// TIA Portal project "PID_controller" (V14)

(* hardware
DEVICE "S71500/ET200MP station_1"  S7-1500 station
   slot 0: "Rail_0"  Rack  6ES7 590-1***0-0AA0
   slot 1: "SERVER_PID"  CPU 1512C-1 PN  6ES7 512-1CK00-0AB0  V2.1
      slot 3: "CPU display_1"  6ES7591-1AA00-0AA0
DEVICE "PID_HMI"  KTP700 Basic PN
   slot 0: "KTP700 Basic PN"  KTP700 Basic PN  6AV2 123-2GB03-0AX0  14.0.1.0
   slot 1: "HMI_RT_1"  KTP700 Basic PN  6AV2 123-2GB03-0AX0  14.0.1.0
   slot 5: "PID_HMI.IE_CP_1"  PROFINET Interface  14.0.1.0
      slot 1: "PROFINET Interface_1"  PROFINET Interface
         slot 1: "Port_1"  Port
*)

// ===== PLC "SERVER_PID"  CPU 1512C-1 PN =====

VAR_GLOBAL   // PLC tag table "Default tag table"
   "Temperature_input" AT %IW0 : Int;
   "Pump_out" AT %QW0 : Int;
END_VAR

DATA_BLOCK "Temperature"   // DB2
{ S7_Optimized_Access := 'TRUE' }
VERSION : 0.1
   VAR
      Temperature_input : Real;
      Temperature_out : Real;
   END_VAR
BEGIN
END_DATA_BLOCK

DATA_BLOCK "PID_DB"   // DB3
{ S7_Optimized_Access := 'TRUE' }
VERSION : 0.1
   VAR
      PID_Setpoint : Real;
      PID_Output : Real;
      PIT_Output_PER : Int;
      PId_Output_PWM : Bool;
      PID_State : Int;
      PID_Error : Bool;
      PID_ModeActivate : Bool;
      PID_manualEnable : Bool;
      PID_ErrorBits : Word;
   END_VAR
BEGIN
END_DATA_BLOCK

DATA_BLOCK "input_PLC_DB"   // DB4
{ S7_Optimized_Access := 'TRUE' }
VERSION : 0.1
// stored: InstanceOfName input_PLC
"input_PLC"
BEGIN
END_DATA_BLOCK

DATA_BLOCK "Pump_freuenceHz"   // DB5
{ S7_Optimized_Access := 'TRUE' }
VERSION : 0.1
   VAR
      Pump_scale : Real;
   END_VAR
BEGIN
END_DATA_BLOCK

FUNCTION_BLOCK "input_PLC"   // FB1, LAD
{ S7_Optimized_Access := 'TRUE' }
VERSION : 0.1
   VAR_INPUT
      input_plc : Real;
   END_VAR
   VAR_OUTPUT
      In_out_DB : Real;
   END_VAR
BEGIN

REGION Network 1
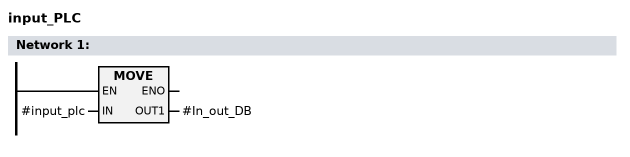
   RUNG wire#powerrail
      Move(in := #input_plc, out1 => #In_out_DB)
   END_RUNG
   // the same network as SCL:
   #In_out_DB := #input_plc;
END_REGION
END_FUNCTION_BLOCK

FUNCTION "analog_input" : Void   // FC1, LAD
{ S7_Optimized_Access := 'TRUE' }
VERSION : 0.1
   VAR_INPUT
      Inpit_min : Int;
      input_max : Int;
      Process_value : Real;
   END_VAR
   VAR_OUTPUT
      Scale_value_out : Real;
   END_VAR
   VAR_TEMP
      temp_value : Real;
   END_VAR
BEGIN

REGION Network 1
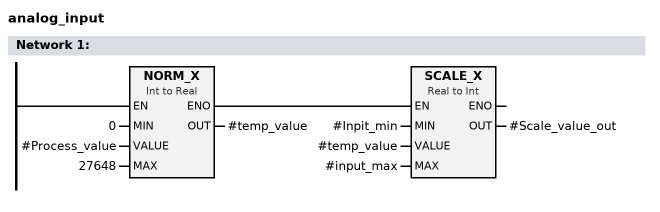
   RUNG wire#powerrail
      { S7_Templates := "[SrcType := Int, DestType := Real]" } Normalize(min := 0, value := #Process_value, max := 27648, out => #temp_value)
      { S7_Templates := "[SrcType := Real, DestType := Int]" } Scale(min := #Inpit_min, value := #temp_value, max := #input_max, out => #Scale_value_out)
   END_RUNG
   // the same network as SCL:
   #temp_value := NORM_X(MIN := 0, VALUE := #Process_value, MAX := 27648);
   #Scale_value_out := SCALE_X(MIN := #Inpit_min, VALUE := #temp_value, MAX := #input_max);
END_REGION
END_FUNCTION

ORGANIZATION_BLOCK "Main"   // OB1, LAD, ProgramCycle
TITLE = "Main Program Sweep (Cycle)"
{ S7_Optimized_Access := 'TRUE' }
VERSION : 0.1
   VAR_INPUT
      Initial_Call : Bool;   // Initial call of this OB
      Remanence : Bool;   // =True, if remanent data are available
   END_VAR
BEGIN

REGION Network 1
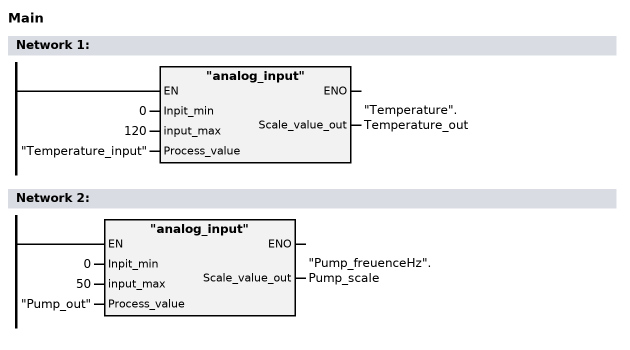
   RUNG wire#powerrail
      "analog_input"(Inpit_min := 0, input_max := 120, Process_value := "Temperature_input", Scale_value_out => "Temperature".Temperature_out)
   END_RUNG
   // the same network as SCL:
   "analog_input"(Inpit_min := 0,
                  input_max := 120,
                  Process_value := "Temperature_input",
                  Scale_value_out => "Temperature".Temperature_out);
END_REGION

REGION Network 2
   RUNG wire#powerrail
      "analog_input"(Inpit_min := 0, input_max := 50, Process_value := "Pump_out", Scale_value_out => "Pump_freuenceHz".Pump_scale)
   END_RUNG
   // the same network as SCL:
   "analog_input"(Inpit_min := 0,
                  input_max := 50,
                  Process_value := "Pump_out",
                  Scale_value_out => "Pump_freuenceHz".Pump_scale);
END_REGION
END_ORGANIZATION_BLOCK

ORGANIZATION_BLOCK "Cyclic interrupt"   // OB30, LAD, CyclicInterrupt
{ S7_Optimized_Access := 'TRUE' }
VERSION : 0.1
   VAR_INPUT
      Initial_Call : Bool;   // Initial call of this OB
      Event_Count : Int;   // Events discarded
   END_VAR
BEGIN

REGION Network 1
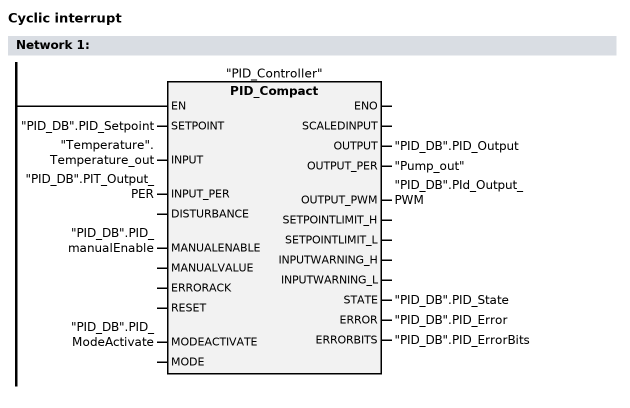
   "PID_Controller"(Setpoint := "PID_DB".PID_Setpoint,   // PID_Compact
                    Input := "Temperature".Temperature_out,
                    Input_PER := "PID_DB".PIT_Output_PER,
                    ManualEnable := "PID_DB".PID_manualEnable,
                    ModeActivate := "PID_DB".PID_ModeActivate,
                    Output => "PID_DB".PID_Output,
                    Output_PER => "Pump_out",
                    Output_PWM => "PID_DB".PId_Output_PWM,
                    State => "PID_DB".PID_State,
                    Error => "PID_DB".PID_Error,
                    ErrorBits => "PID_DB".PID_ErrorBits);
END_REGION
END_ORGANIZATION_BLOCK

(* ===== HMI "HMI_RT_1" =====
system functions are stored by id; their names below are inferred from use
connection "HMI_Connection_1": ETHERNET, SMART_S7_1500_OMS

HMI tags "Default tag table"
   "Tag_ScreenNumber" : UInt, internal
   "PID_DB_PID_Setpoint" : Real = PLC PID_DB.PID_Setpoint, 1 s
   "Temperature_Temperature_out" : Real = PLC Temperature.Temperature_out, 1 s
   "Pump_freuenceHz_Pump_scale" : Real = PLC Pump_freuenceHz.Pump_scale, 1 s
   "PID_DB_PID_ModeActivate" : Bool = PLC PID_DB.PID_ModeActivate, 1 s
   "PID_DB_PID_Output" : Real = PLC PID_DB.PID_Output, 1 s

Template "Template_1" 800x480
   SymbolicIOField "Symbolic_IO_Field_Screen" at 93,9 size 600x33; TextOff '0'; TextOn '1'; TextList "TextList_ScreenNames"
      ProcessValue <- "Tag_ScreenNumber"
      on Change: ActivateScreenByNumber("Tag_ScreenNumber", 0)
   DateTimeField "HmiScreenItemData" at 695,25 size 105x25
   DateTimeField "HmiScreenItemData_1" at 695,0 size 105x25
   GraphicView "Logo" at 0,0 size 91x51; Picture "Logo of HMI_1"

screen "Root screen" 800x480, template "Template_1"
   on GenerateScreen: SetTag("Tag_ScreenNumber", 1)
   TextField "Text field_1" at 101,52 size 86x25; Text 'Enable PID'
   Button "Button_1" at 38,77 size 96x32; TextOff 'Enable'
      on Press: SetBit("PID_DB_PID_ModeActivate")
   Button "Button_2" at 38,123 size 96x32; TextOff 'Disable'
      on Release: ResetBit("PID_DB_PID_ModeActivate")
   TextField "Text field_2" at 550,52 size 93x25; Text 'Controll PID'
   TextField "Text field_3" at 456,77 size 111x25; Text 'Setpoint Value'
   TextField "Text field_4" at 456,109 size 107x25; Text 'Prosess Value'
   TextField "Text field_5" at 456,141 size 95x25; Text 'Pump Speed'
   IOField "I/O field_2" at 626,77 size 96x32; FormatPattern 9999.99
      ProcessValue <- "PID_DB_PID_Setpoint"
   IOField "I/O field_3" at 626,114 size 96x32; FormatPattern 9999.99
      ProcessValue <- "Temperature_Temperature_out"
   IOField "I/O field_4" at 626,150 size 96x32; FormatPattern 9999.99
      ProcessValue <- "Pump_freuenceHz_Pump_scale"
   TrendView "Trend view_1" at 8,194 size 784x278
   GraphicView "Graphic view_1" at 208,52 size 141x107; Picture "Graphic_1"
   Rectangle "Rectangle_3" at 256,102 size 55x29
      Appearance <- "PID_DB_PID_ModeActivate"
*)